GLOBALCONSTANTS OPC_Strings (* Global constants *)
  (* Standard: 61499-1; Description: Copyright (c) 2026 Meisterschulen am Ostbahnhof This program and the accompanying materials are made available under the terms of the Eclipse Public License 2.0 which is available at https://www.eclipse.org/legal/epl-2.0/ SPDX-License-Identifier: EPL-2.0 *)
  (* Version 1.0, 2026-08-31, Franz Höpfinger, Meisterschulen am Ostbahnhof *)
  PACKAGE Uebungen::const::OPC;
  VAR_GLOBAL CONSTANT
    Uebung12h_READ : WSTRING := "opc_ua[READ;/Objects/Uebung12h/VALUE,1:s=Uebung12h_VALUE]";
    Uebung12h_WRITE : WSTRING := "opc_ua[WRITE;/Objects/Uebung12h/VALUE,1:s=Uebung12h_VALUE]";
    Uebung12i_READ : WSTRING := "opc_ua[READ;/Objects/Uebung12i/VALUE,1:s=Uebung12i_VALUE]";
    Uebung12i_WRITE : WSTRING := "opc_ua[WRITE;/Objects/Uebung12i/VALUE,1:s=Uebung12i_VALUE]";
    Uebung12n_READ : WSTRING := "opc_ua[READ;/Objects/Uebung12n/VALUE,1:s=Uebung12n_VALUE]";
    Uebung12n_WRITE : WSTRING := "opc_ua[WRITE;/Objects/Uebung12n/VALUE,1:s=Uebung12n_VALUE]";
    Uebung12o_READ : WSTRING := "opc_ua[READ;/Objects/Uebung12o/VALUE,1:s=Uebung12o_VALUE]";
    Uebung12o_WRITE : WSTRING := "opc_ua[WRITE;/Objects/Uebung12o/VALUE,1:s=Uebung12o_VALUE]";
  END_VAR
END_GLOBALCONSTANTS
